FUNCTION_BLOCK GreenMasterAIU_ModbusRTU EXTENDS GreenMasterAIU_Base
VAR_INPUT
END_VAR
VAR_OUTPUT
END_VAR
VAR
	ModbusRTU: ModbusRTU;
	ModbusWord_T_BF1: ModbusReadWord;
	ModbusWord_F_BF1: ModbusReadWord;
	ModbusWord_T_BP1: ModbusReadWord;
	ModbusWord_F_BP1: ModbusReadWord;
	ModbusWord_T_BP2: ModbusReadWord;
	ModbusWord_F_BP2: ModbusReadWord;
	ModbusWord_F_BP3: ModbusReadWord;
	IO_AI_T_BP1: PressureInput;
	IO_AI_F_BP1: PressureInput;
	IO_AI_T_BP2: PressureInput;
	IO_AI_F_BP2: PressureInput;
	IO_AI_F_BP3: PressureInput;
	IO_AI_T_BF1: FlowInput;
	IO_AI_F_BF1: FlowInput;
END_VAR


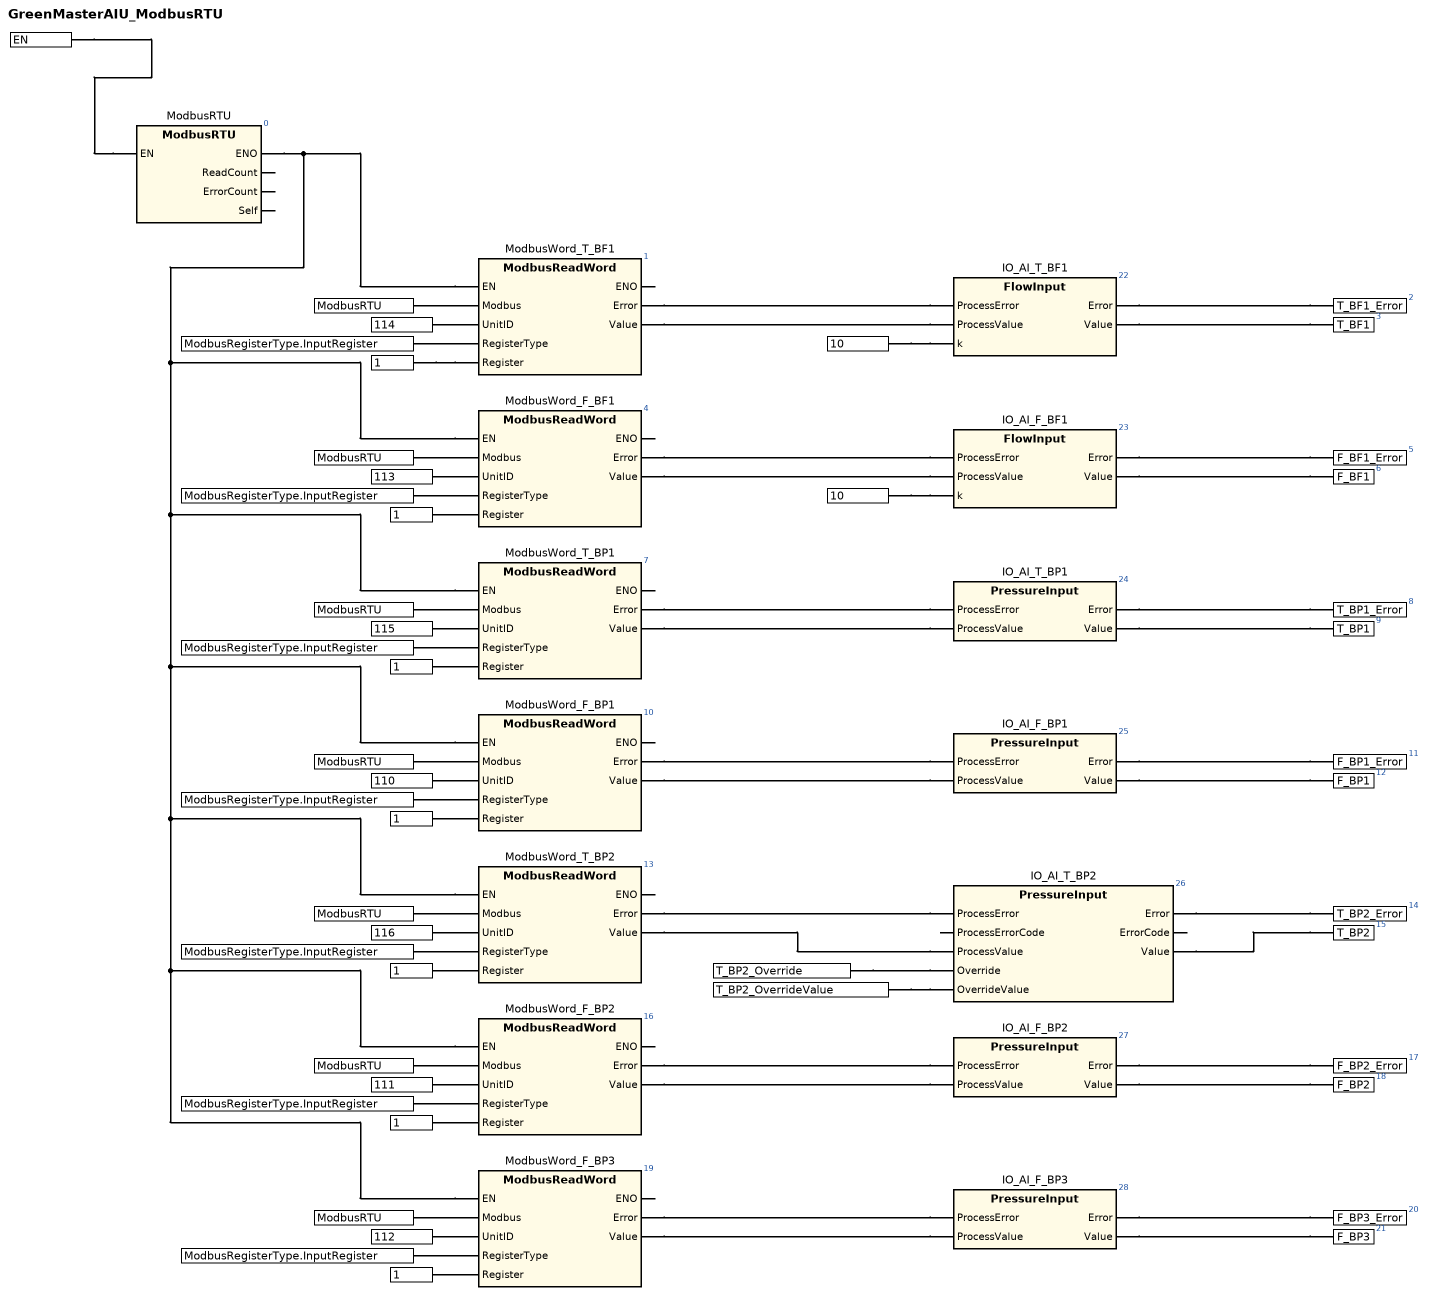
// PAGE
ModbusRTU(EN := EN);
ModbusWord_T_BF1(
    EN := ModbusRTU.ENO,
    Modbus := ModbusRTU,
    UnitID := 114,
    RegisterType := ModbusRegisterType.InputRegister,
    Register := 1); // ModbusReadWord
T_BF1_Error := IO_AI_T_BF1.Error;
T_BF1 := IO_AI_T_BF1.Value;
ModbusWord_F_BF1(
    EN := ModbusRTU.ENO,
    Modbus := ModbusRTU,
    UnitID := 113,
    RegisterType := ModbusRegisterType.InputRegister,
    Register := 1); // ModbusReadWord
F_BF1_Error := IO_AI_F_BF1.Error;
F_BF1 := IO_AI_F_BF1.Value;
ModbusWord_T_BP1(
    EN := ModbusRTU.ENO,
    Modbus := ModbusRTU,
    UnitID := 115,
    RegisterType := ModbusRegisterType.InputRegister,
    Register := 1); // ModbusReadWord
T_BP1_Error := IO_AI_T_BP1.Error;
T_BP1 := IO_AI_T_BP1.Value;
ModbusWord_F_BP1(
    EN := ModbusRTU.ENO,
    Modbus := ModbusRTU,
    UnitID := 110,
    RegisterType := ModbusRegisterType.InputRegister,
    Register := 1); // ModbusReadWord
F_BP1_Error := IO_AI_F_BP1.Error;
F_BP1 := IO_AI_F_BP1.Value;
ModbusWord_T_BP2(
    EN := ModbusRTU.ENO,
    Modbus := ModbusRTU,
    UnitID := 116,
    RegisterType := ModbusRegisterType.InputRegister,
    Register := 1); // ModbusReadWord
T_BP2_Error := IO_AI_T_BP2.Error;
T_BP2 := IO_AI_T_BP2.Value;
ModbusWord_F_BP2(
    EN := ModbusRTU.ENO,
    Modbus := ModbusRTU,
    UnitID := 111,
    RegisterType := ModbusRegisterType.InputRegister,
    Register := 1); // ModbusReadWord
F_BP2_Error := IO_AI_F_BP2.Error;
F_BP2 := IO_AI_F_BP2.Value;
ModbusWord_F_BP3(
    EN := ModbusRTU.ENO,
    Modbus := ModbusRTU,
    UnitID := 112,
    RegisterType := ModbusRegisterType.InputRegister,
    Register := 1); // ModbusReadWord
F_BP3_Error := IO_AI_F_BP3.Error;
F_BP3 := IO_AI_F_BP3.Value;
IO_AI_T_BF1(ProcessError := ModbusWord_T_BF1.Error, ProcessValue := ModbusWord_T_BF1.Value, k := 10); // FlowInput
IO_AI_F_BF1(ProcessError := ModbusWord_F_BF1.Error, ProcessValue := ModbusWord_F_BF1.Value, k := 10); // FlowInput
IO_AI_T_BP1(ProcessError := ModbusWord_T_BP1.Error, ProcessValue := ModbusWord_T_BP1.Value); // PressureInput
IO_AI_F_BP1(ProcessError := ModbusWord_F_BP1.Error, ProcessValue := ModbusWord_F_BP1.Value); // PressureInput
IO_AI_T_BP2(
    ProcessError := ModbusWord_T_BP2.Error,
    ProcessValue := ModbusWord_T_BP2.Value,
    Override := T_BP2_Override,
    OverrideValue := T_BP2_OverrideValue); // PressureInput
IO_AI_F_BP2(ProcessError := ModbusWord_F_BP2.Error, ProcessValue := ModbusWord_F_BP2.Value); // PressureInput
IO_AI_F_BP3(ProcessError := ModbusWord_F_BP3.Error, ProcessValue := ModbusWord_F_BP3.Value); // PressureInput

END_FUNCTION_BLOCK

(* stored: Version 1.1.0.1, ProductVersion 3.1.4024.6
   POU GreenMasterAIU_ModbusRTU: Id {b6854a93-3767-453a-af2d-d9c9f71d6792}, SpecialFunc None *)
